{attribute wpf [Container(Layout.Border)]}
TYPE BorderLayout:
STRUCT
	_various_types: VariousTypes;
END_STRUCT
END_TYPE

(* stored: Version 1.1.0.1, ProductVersion 3.1.4024.9
   DUT BorderLayout: Id {85daafbc-697a-49c1-8928-6d5fe9743da9} *)
